DATA_BLOCK "Werkskreislauf_DB"
{ S7_Optimized_Access := 'TRUE' }
VERSION : 0.1
NON_RETAIN
"Werkskreislauf"

BEGIN

END_DATA_BLOCK

